PROGRAM HMI
VAR
	astHmiControl: ARRAY [1..GVL_APP.nAXIS_NUM] OF ST_HmiControl;
	eHmiControl : E_HmiControl;
	eSWLimitControl : E_SWLimitControl;
	iHmiAxisSelection : INT;
	iKeyPressedValue : INT := -1;
	iSelectedAxis : INT := -1;
	aiUsedKeys : ARRAY[1..12] OF INT := [E_HmiControl.JogFwd, E_HmiControl.JogBwd,
    E_HmiControl.SmallTweakFwd, E_HmiControl.SmallTweakBwd, E_HmiControl.MediumTweakFwd, 
	E_HmiControl.MediumTweakBwd, E_HmiControl.BigTweakFwd, E_HmiControl.BigTweakBwd, 
	E_HmiControl.AbsMove, E_HmiControl.Stop, E_HmiControl.SlowJogFwd, E_HmiControl.SlowJogBwd];
	iUsedKeysIndex : INT;
	iSmallTweakDistance : REAL := 0.1;	
	iMediumTweakDistance : REAL := 1;
	iBigTweakDistance : REAL := 5;
	iHmiAxisCounter : INT;
	bResetParameters : BOOL := FALSE;
	
	bLocalMode: BOOL;
	fbLocalModeRTrig: R_TRIG;
	fbLocalModeFTrig: F_TRIG;
	
	bSWLimitsOn : BOOL := FALSE; //False for off, true for on
END_VAR

bLocalMode:= SAFETY.inLocalMode;
fbLocalModeRTrig(CLK := bLocalMode);
fbLocalModeFTrig(CLK := bLocalMode);

IF bResetParameters THEN
	ResetParameters();
END_IF


IF ketop.keys[E_HmiControl.Stop] OR NOT bLocalMode THEN
	eHmiControl := E_HmiControl.Stop;
END_IF


CASE eHmiControl OF
	E_HmiControl.Default:
		iKeyPressedValue := -1;
		iSelectedAxis := -1;
		IF iHmiAxisSelection > 0 AND iHmiAxisSelection <= UINT_TO_INT(GVL_APP.nAXIS_NUM) THEN
			FOR iUsedKeysIndex := 1 TO (SIZEOF(aiUsedKeys)/SIZEOF(UINT)) DO
				IF KeTop.keys[aiUsedKeys[iUsedKeysIndex]] = TRUE THEN
					iKeyPressedValue := aiUsedKeys[iUsedKeysIndex];
					iSelectedAxis := iHmiAxisSelection;
					eHmiControl := iKeyPressedValue;
				END_IF
			END_FOR
		END_IF
		
	E_HmiControl.JogFwd:
		astAxes[iSelectedAxis].stControl.fVelocity := ABS(astAxes[iSelectedAxis].stControl.fVelocity);
		Jog(fOverride:= astHmiControl[iSelectedAxis].fVelocity);
		eHmiControl := E_HmiControl.WaitForJogFinish;
	
	E_HmiControl.JogBwd:
		astAxes[iSelectedAxis].stControl.fVelocity := -ABS(astAxes[iSelectedAxis].stControl.fVelocity);
		Jog(fOverride:= astHmiControl[iSelectedAxis].fVelocity);
		eHmiControl := E_HmiControl.WaitForJogFinish;
		
	E_HmiControl.SlowJogFwd:
		astAxes[iSelectedAxis].stControl.fVelocity := ABS(astAxes[iSelectedAxis].stControl.fVelocity);
		Jog(fOverride:= 0.2*astHmiControl[iSelectedAxis].fVelocity);
		eHmiControl := E_HmiControl.WaitForJogFinish;		
		
	E_HmiControl.SlowJogBwd:
		astAxes[iSelectedAxis].stControl.fVelocity := -ABS(astAxes[iSelectedAxis].stControl.fVelocity);
		Jog(fOverride:= 0.2*astHmiControl[iSelectedAxis].fVelocity);
		eHmiControl := E_HmiControl.WaitForJogFinish;	
	
	E_HmiControl.WaitForJogFinish:
		IF Ketop.keys[iKeyPressedValue] = FALSE THEN
			astAxes[iSelectedAxis].stControl.bHalt := TRUE;
			astAxes[iSelectedAxis].stControl.fVelocity := ABS(astAxes[iSelectedAxis].stControl.fVelocity);
			eHmiControl := E_HmiControl.Default;
		END_IF

	E_HmiControl.SmallTweakFwd:
		Tweak(iSmallTweakDistance);
		eHmiControl := E_HmiControl.WaitForTweakFinish;

	E_HmiControl.SmallTweakBwd:
		Tweak(-iSmallTweakDistance);
		eHmiControl := E_HmiControl.WaitForTweakFinish;
	
	E_HmiControl.MediumTweakFwd:
		Tweak(iMediumTweakDistance);
		eHmiControl := E_HmiControl.WaitForTweakFinish;

	E_HmiControl.MediumTweakBwd:
		Tweak(-iMediumTweakDistance);
		eHmiControl := E_HmiControl.WaitForTweakFinish;
		
	E_HmiControl.BigTweakFwd:
		Tweak(iBigTweakDistance);
		eHmiControl := E_HmiControl.WaitForTweakFinish;

	E_HmiControl.BigTweakBwd:
		Tweak(-iBigTweakDistance);
		eHmiControl := E_HmiControl.WaitForTweakFinish;
		
	E_HmiControl.WaitForTweakFinish:
		IF Ketop.keys[iKeyPressedValue] = FALSE AND astAxes[iSelectedAxis].stStatus.bMoving = FALSE THEN
			eHmiControl := E_HmiControl.Default;
		END_IF
		
	E_HmiControl.AbsMove:
		astAxes[iSelectedAxis].stConfig.fOverride := astHmiControl[iSelectedAxis].fVelocity;
		astAxes[iSelectedAxis].stControl.fPosition := astHmiControl[iSelectedAxis].fTargetPosition;
		astAxes[iSelectedAxis].stControl.eCommand := E_MotionFunctions.eLocalMoveAbsolute;
		astAxes[iSelectedAxis].stControl.bExecute := TRUE; 
		eHmiControl := E_HmiControl.WaitForAbsoluteFinish;
	
	E_HmiControl.WaitForAbsoluteFinish:
		IF astAxes[iSelectedAxis].stStatus.bMoving = FALSE THEN
			eHmiControl := E_HmiControl.Default;	
		END_IF
	
	E_HmiControl.Stop:
		IF iSelectedAxis > 0 THEN
			astAxes[iSelectedAxis].stControl.bHalt := TRUE;
			IF ketop.keys[E_HmiControl.Stop] = FALSE AND astAxes[iSelectedAxis].stStatus.bMoving = FALSE THEN
				eHmiControl := E_HmiControl.Default;
				FOR iUsedKeysIndex := 1 TO (SIZEOF(aiUsedKeys)/SIZEOF(UINT)) DO
					IF KeTop.keys[aiUsedKeys[iUsedKeysIndex]] = TRUE THEN
						eHmiControl := E_HmiControl.Stop;
					END_IF
				END_FOR
			END_IF	
		END_IF
		IF iSelectedAxis = -1 AND bLocalMode THEN
			eHmiControl := E_HmiControl.Default;
		END_IF

END_CASE

CASE eSWLimitControl OF
	E_SWLimitControl.Default:
		IF fbLocalModeRTrig.Q THEN
			//eSWLimitControl := E_SWLimitControl.EnableSWLimits;
		END_IF
		IF fbLocalModeFTrig.Q THEN
			eSWLimitControl := E_SWLimitControl.DisableSWLimits;
		END_IF
	
	E_SWLimitControl.EnableSWLimits:
		bSWLimitsOn := TRUE;
		KeTop.screenBrightness := 100;
		FOR iHmiAxisCounter := 1 TO GVL_APP.nAXIS_NUM DO
			ToggleSWLimits();	
		END_FOR
		eSWLimitControl := E_SWLimitControl.Default;
	
	E_SWLimitControl.DisableSWLimits:
		bSWLimitsOn := FALSE;
		FOR iHmiAxisCounter := 1 TO GVL_APP.nAXIS_NUM DO
			ToggleSWLimits();	
		END_FOR
		eSWLimitControl := E_SWLimitControl.Default;
	
	E_SWLimitControl.WriteFwdLimit:
		IF bLocalMode THEN
			astAxes[iHmiAxisSelection].stConfig.eAxisParameters := E_AxisParameters.SWLimitForward;
			astAxes[iHmiAxisSelection].stConfig.fWriteAxisParameter := astHmiControl[iHmiAxisSelection].fFwdLimit;
			WriteToSWLimit();
		END_IF
		eSWLimitControl := E_SWLimitControl.Default;
	
	E_SWLimitControl.WriteBwdLimit:
		IF bLocalMode THEN
			astAxes[iHmiAxisSelection].stConfig.eAxisParameters := E_AxisParameters.SWLimitBackward;
			astAxes[iHmiAxisSelection].stConfig.fWriteAxisParameter := astHmiControl[iHmiAxisSelection].fBwdLimit;
			WriteToSWLimit();	
		END_IF
		eSWLimitControl := E_SWLimitControl.Default;
	
END_CASE

METHOD Jog
VAR_INPUT
	fOverride : LREAL;
END_VAR
astAxes[iSelectedAxis].stConfig.fOverride := fOverride;
astAxes[iSelectedAxis].stControl.eCommand:= E_MotionFunctions.eLocalMoveVelocity;
astAxes[iSelectedAxis].stControl.bExecute:= TRUE;
END_METHOD

ACTION ResetParameters:
FOR iHmiAxisCounter := 1 TO GVL_APP.nAXIS_NUM DO
	astHmiControl[iHmiAxisCounter].fTargetPosition := 0;
	astHmiControl[iHmiAxisCounter].fVelocity := 100;	
END_FOR
bResetParameters := FALSE;
END_ACTION

ACTION ToggleSWLimits:
astAxes[iHmiAxisCounter].stControl.eCommand := E_MotionFunctions.eWriteToggleSWLimits;
astAxes[iHmiAxisCounter].stConfig.fWriteAxisBoolParameter := bSWLimitsOn;
astAxes[iHmiAxisCounter].stControl.bExecute := TRUE;
END_ACTION

METHOD Tweak
VAR_INPUT
	TweakDistance : LREAL;
END_VAR
astAxes[iSelectedAxis].stConfig.fOverride :=100;
astAxes[iSelectedAxis].stControl.fRelativePosition := TweakDistance;
astAxes[iSelectedAxis].stControl.eCommand:=E_MotionFunctions.eLocalMoveRelative;
astAxes[iSelectedAxis].stControl.bExecute:=TRUE;
END_METHOD

ACTION WriteToSWLimit:
astAxes[iHmiAxisSelection].stControl.eCommand := E_MotionFunctions.eWriteParameter;
astAxes[iHmiAxisSelection].stControl.bExecute := TRUE;
END_ACTION

END_PROGRAM

(* stored: Version 1.1.0.1, ProductVersion 3.1.4026.18
   POU HMI: Id {059d275e-4870-4167-960e-2a5c721e374f}, SpecialFunc None
   Method Jog: Id {1ac9d73a-3fde-4d7c-ab9f-a89280ff125b}
   Action ResetParameters: Id {ede581f7-17f2-47ed-bf91-d81c7a0e26c6}
   Action ToggleSWLimits: Id {00f2d6f2-ec9f-43a1-b3f7-222658b8123f}
   Method Tweak: Id {7c4ad566-6209-4d9e-849a-b4a915c383eb}
   Action WriteToSWLimit: Id {a474f6c3-01a0-4eec-83a2-dbe3d219df3f} *)
